(*			
	EVERDE sp. z o.o.
	Rafał Osajda		21.08.2025		TC 4024.66
	Interfejs łaczący na potrzeby przekazania do elementu
*)
INTERFACE ITF_Electrovalve_HMI_Init EXTENDS ITF_BaseComponent, ITF_Electrovalve_HMI_Connector

END_INTERFACE

(* stored: Version 1.1.0.1
   Itf ITF_Electrovalve_HMI_Init: Id {b4f18e5e-f2cb-4769-94d5-7abeb274cb1f} *)
